Staubli VAL3: oSample.pgx

public program oSample(num nChoice (dimensions=1))
// oSample
begin
  dioSet(oSample,nChoice)
end
